// TIA Portal project "Masterprojekt" (V14)

(* hardware
DEVICE "S71500/ET200MP-Station_1"  S7-1500 station
   slot 0: "Profilschiene_0"  Rack  6ES7 590-1***0-0AA0
   slot 1: "PLC_1"  CPU 1512C-1 PN  6ES7 512-1CK00-0AB0  V2.0
      slot 3: "CPU-Display_1"  6ES7591-1AA00-0AA0
*)

// ===== PLC "PLC_1"  CPU 1512C-1 PN =====

DATA_BLOCK "Datenbaustein_1"   // DB1
{ S7_Optimized_Access := 'FALSE' }
VERSION : 0.1
   VAR
      orderID : DInt;
      orderCompleted : Bool := true;
      timeOrderCompleted : DTL;
      orderName : Array[0..63] of Char;
      heightA1 : Byte;
      heightA2 : Byte;
      heightA3 : Byte;
      heightA4 : Byte;
      heightA5 : Byte;
      heightB1 : Byte;
      heightB2 : Byte;
      heightB3 : Byte;
      heightB4 : Byte;
      heightB5 : Byte;
      productionStock15mmSilver : Byte;
      productionStock15mmBlue : Byte;
      productionStock18mmSilver : Byte;
      productionStock18mmBlue : Byte;
      productionStock22mmSilver : Byte;
      productionStock22mmBlue : Byte;
   END_VAR
BEGIN
END_DATA_BLOCK